PROGRAM MAIN
VAR
	eEventType1 : E_Event := E_Event.Warning;
	eEventSeverity1 : TcEventSeverity := TcEventSeverity.Critical;
	nEventIdentity1 : UDINT := 32;
	sEventText1 : STRING(255) :=  'This is a danger';
	
	EventLogger1 : EventLogger;
	fbMotor1 : Motor;
	
	nNum1 : INT;
	nNum2 : INT := 43;
	nSum : INT;
	
	nMotorValue1 : DINT;
	nMotorValue2 : DINT;
	bMotorRunning : BOOL;
	
	bFlag : BOOL := TRUE;
END_VAR

IF bFlag THEN
	EventLogger1.AddItem(eEventType:= eEventType1,eEventSeverity := eEventSeverity1,nEventIdentity := nEventIdentity1,sEventText := sEventText1 );
	GVL_Sum.nNumber1 := GVL_Sum.nNumber1 + 1;
	nMotorValue1 := fbMotor1.nMotorValue;
	fbMotor1();
	nMotorValue2 := fbMotor1.nMotorValue;
	nSum := AddNums(fbMotor1);
	
	bFlag := FALSE;
END_IF

END_PROGRAM

(* stored: Version 1.1.0.1, ProductVersion 3.1.4024.16
   POU MAIN: Id {6acb3596-614b-4bd6-88d1-a625d8d1eebd}, SpecialFunc None *)
